{attribute addProperty BoxType "EJ2502-0000-0023"}
{attribute addProperty Id "PWM_outputAT %Q*UINT162"}
{attribute addProperty CRC "2822587050"}
{attribute addProperty SizeInBites "16"}
{attribute addProperty SizeInBytes "2"}
TYPE PWM_Outputs_Channel_A83D42AA :
STRUCT
	{attribute addProperty Name "PWM_output"}
	PWM_output AT %Q* : UINT;
END_STRUCT
END_TYPE

(* stored: Version 1.2.0.0, ProductVersion 3.1.4024.9
   DUT PWM_Outputs_Channel_A83D42AA: Id {d948ffe4-f9a5-4851-befd-5b4d699d9b88} *)
